(* CoDeSys 2.3.9.26 project: Q.pro *)
(* Libraries: Util.lib 18.5.10 23:14:28, Standard.LIB 4.10.05 19:14:46 *)

(* POU PLC_PRG, LD *)
PROGRAM PLC_PRG
VAR

	M4000: BOOL;		(*Internal Safety Relay*)
	PBONOFF: BOOL;		(*ON/OFF*)
	PBEstop: BOOL;		(*E-Stop*)
	H1: BOOL;		(*T1 High Limit*)
	H2: BOOL;		(*T2 High Limit*)
	Alarm: BOOL;
	Start: BOOL;
	R1: BOOL;
	Stop: BOOL;
	Reset: BOOL;
	Ready: BOOL;
	R0: BOOL;
	Pump01: BOOL;
	V1: BOOL;		(*Valve 1*)
	M1: BOOL;
	R2: INT := 0;
	L1: BOOL;
END_VAR
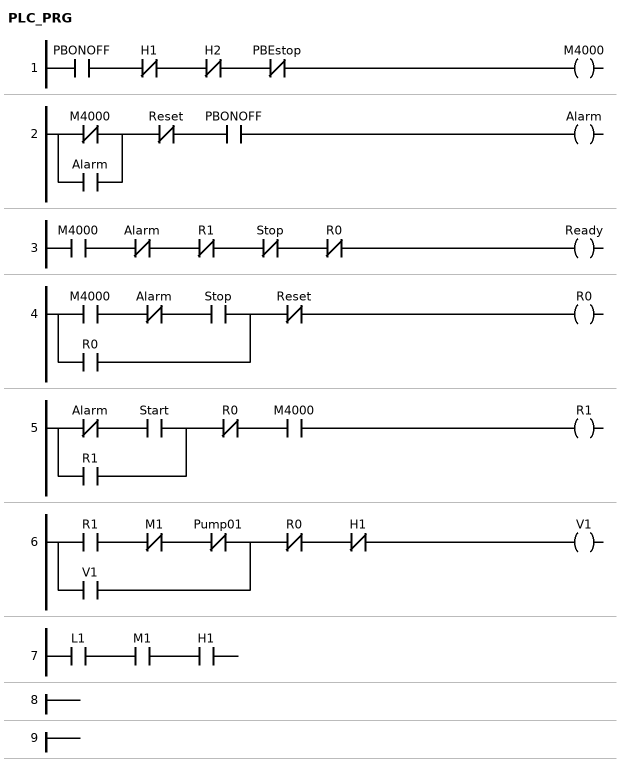
_LD_ (* Ladder Diagram *)
NETWORK 1
	[PBONOFF] - [/H1] - [/H2] - [/PBEstop] --- (M4000)
NETWORK 2
	{ [/M4000] | [Alarm] } - [/Reset] - [PBONOFF] --- (Alarm)
NETWORK 3
	[M4000] - [/Alarm] - [/R1] - [/Stop] - [/R0] --- (Ready)
NETWORK 4
	{ [M4000] - [/Alarm] - [Stop] | [R0] } - [/Reset] --- (R0)
NETWORK 5
	{ [/Alarm] - [Start] | [R1] } - [/R0] - [M4000] --- (R1)
NETWORK 6
	{ [R1] - [/M1] - [/Pump01] | [V1] } - [/R0] - [/H1] --- (V1)
NETWORK 7
	[L1] - [M1] - [H1]
NETWORK 8
	*
NETWORK 9
	*
_END_LD_
(* the same logic as Structured Text *)
(* Network 1 *)
M4000 := PBONOFF AND NOT H1 AND NOT H2 AND NOT PBEstop;
(* Network 2 *)
Alarm := (NOT M4000 OR Alarm) AND NOT Reset AND PBONOFF;
(* Network 3 *)
Ready := M4000 AND NOT Alarm AND NOT R1 AND NOT Stop AND NOT R0;
(* Network 4 *)
R0 := (M4000 AND NOT Alarm AND Stop OR R0) AND NOT Reset;
(* Network 5 *)
R1 := (NOT Alarm AND Start OR R1) AND NOT R0 AND M4000;
(* Network 6 *)
V1 := (R1 AND NOT M1 AND NOT Pump01 OR V1) AND NOT R0 AND NOT H1;
(* Network 7 *)
(* Network 8 *)
(* Network 9 *)
END_PROGRAM

(* Visualisation HMI
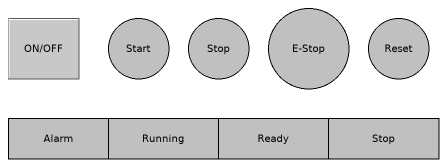
ellipse at (130,20)-(191,81): text "Start"; alarm colour if PLC_PRG.Start; taps PLC_PRG.Start
ellipse at (210,20)-(271,81): text "Stop"; alarm colour if PLC_PRG.Stop; taps PLC_PRG.Stop
ellipse at (290,10)-(371,91): text "E-Stop"; alarm colour if PLC_PRG.PBEstop; toggles PLC_PRG.PBEstop
ellipse at (390,20)-(451,81): text "Reset"; taps PLC_PRG.Reset
rectangle at (30,120)-(131,161): text "Alarm"; alarm colour if PLC_PRG.Alarm
rectangle at (130,120)-(241,161): text "Running"; alarm colour if PLC_PRG.R1
rectangle at (240,120)-(351,161): text "Ready"; alarm colour if PLC_PRG.Ready
rectangle at (350,120)-(461,161): text "Stop"; alarm colour if PLC_PRG.R0
button at (30,20)-(101,81): text "ON/OFF"; toggles PLC_PRG.PBONOFF
*)

(* Visualisation Machine
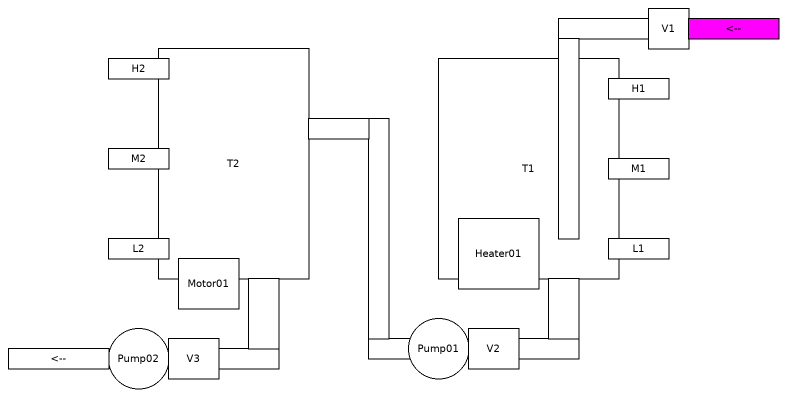
rectangle at (200,60)-(351,291): text "T2"
rectangle at (150,70)-(211,91): text "H2"
rectangle at (150,160)-(211,181): text "M2"
rectangle at (150,250)-(211,271): text "L2"
rectangle at (480,70)-(661,291): text "T1"
rectangle at (600,30)-(691,51): alarm colour if PLC_PRG.V1
rectangle at (650,170)-(711,191): text "M1"
ellipse at (150,340)-(211,401): text "Pump02"
rectangle at (650,90)-(711,111): text "H1"
rectangle at (650,250)-(711,271): text "L1"
rectangle at (600,50)-(621,251): alarm colour if PLC_PRG.V1
rectangle at (690,20)-(731,61): text "V1"; alarm colour if PLC_PRG.V1
ellipse at (450,330)-(511,391): text "Pump01"
rectangle at (510,340)-(561,381): text "V2"
rectangle at (730,30)-(821,51): text "<--"
rectangle at (210,350)-(261,391): text "V3"
rectangle at (50,360)-(151,381): text "<--"
rectangle at (220,270)-(281,321): text "Motor01"
rectangle at (500,230)-(581,301): text "Heater01"
7 more shapes without text or variables
*)
